// TIA Portal V18 export
FUNCTION "AHUFrostProtectionDemand" : Void   // FC60018, LAD
{ S7_Optimized_Access := 'TRUE' }
VERSION : 0.1
// stored: AutoNumber false, IsIECCheckEnabled false, SetENOAutomatically false, UDAEnableTagReadback false
   VAR_INPUT
      UnitID : Int;
      SupplyAirTemp : Real;
      FrostSensorAirTemp : Real;
      FrostSensorWaterTemp : Real;
      FrostTstat : Bool;
      OutdoorAirTemperature : Real;
   END_VAR
   VAR_OUTPUT
      FrostProtectionDemand : Real;
   END_VAR
BEGIN
END_FUNCTION
